PROGRAM MAIN
VAR
END_VAR

END_PROGRAM

(* stored: Version 1.1.0.1
   POU MAIN: Id {9452d847-2247-44a3-ba94-9f58b5af4c44} *)
